{attribute 'qualified_only'}
VAR_GLOBAL CONSTANT
	MAX_BYTE_SIZE : UDINT := 1000;
END_VAR

(* stored: Version 1.1.0.1, ProductVersion 3.1.4020.12
   GVL CollectionParameters: Id {86369202-86a7-4fbe-8930-f6f12b29a3f7}, ParameterList True *)
